(* CODESYS project GVL_MOTION_MANAGER.gvl.xml

Project tree, tasks and I/O mapping:
  global variables GVL_MOTION_MANAGER
*)

// GVL_MOTION_MANAGER
{attribute 'qualified_only'}
VAR_GLOBAL
	stMotionManager : ST_MOTION_MANAGER; // Команды, статусы и диагностика менеджера движения
END_VAR
